// TIA Portal V17 export
// export: Created 2022-07-28T18:03:18.4124527Z, ExportSetting None, DisplayName Totally Integrated Automation Portal, DisplayVersion V17, DisplayName TIA Portal Openness, DisplayVersion V17, DisplayName TIA Portal Teamcenter Gateway, DisplayVersion V17, DisplayName TIA Portal Version Control Interface, DisplayVersion V17, DisplayName TIA Portal Test Suite Advanced, DisplayVersion V17, DisplayName SINAMICS Startdrive Advanced, DisplayVersion V17, DisplayName SINAMICS DCC, DisplayVersion V17, DisplayName SINAMICS Startdrive G130, G150, S120, S150, SINAMICS MV, S210, DisplayVersion V17, DisplayName SINAMICS Startdrive G110M, G120, G120C, G120D, G120P, G115D, DisplayVersion V17, DisplayName STEP 7 Professional, DisplayVersion V17, DisplayName SIMATIC Energy Suite, DisplayVersion V17, DisplayName STEP 7 CFC, DisplayVersion V17, DisplayName STEP 7 Safety, DisplayVersion V17, DisplayName WinCC Advanced / Unified PC, DisplayVersion V17, DisplayName SIMATIC Visualization Architect, DisplayVersion V17
TYPE "_ASensor_AlarmBits"
   STRUCT
      ErrorHH { ExternalAccessible := 'False'; ExternalVisible := 'False'; ExternalWritable := 'False'} : Bool;   // x0 - HH fault is active
      ErrorH { ExternalAccessible := 'False'; ExternalVisible := 'False'; ExternalWritable := 'False'} : Bool;   // x1 - H fault is active
      ErrorL { ExternalAccessible := 'False'; ExternalVisible := 'False'; ExternalWritable := 'False'} : Bool;   // x2 - L fault is active
      ErrorLL { ExternalAccessible := 'False'; ExternalVisible := 'False'; ExternalWritable := 'False'} : Bool;   // x3 - LL fault is active
      ErrorOvershoot { ExternalAccessible := 'False'; ExternalVisible := 'False'; ExternalWritable := 'False'} : Bool;   // x4 - Overshoot is active (act val > Maxlim)
      ErrorHiLimit { ExternalAccessible := 'False'; ExternalVisible := 'False'; ExternalWritable := 'False'} : Bool;   // x5 - Exceeding the maximum
      ErrorLoLimit { ExternalAccessible := 'False'; ExternalVisible := 'False'; ExternalWritable := 'False'} : Bool;   // x6 - Exceeding the minimum
      SimMode { ExternalAccessible := 'False'; ExternalVisible := 'False'; ExternalWritable := 'False'} : Bool;   // x7 - Sim mode is active
      NotSimMode { ExternalAccessible := 'False'; ExternalVisible := 'False'; ExternalWritable := 'False'} : Bool := true;   // x8 - Sim mode disabled
      SupplyErr { ExternalAccessible := 'False'; ExternalVisible := 'False'; ExternalWritable := 'False'} : Bool;   // x9 - Error of supply
      AW1_bit10 { ExternalAccessible := 'False'; ExternalVisible := 'False'; ExternalWritable := 'False'} : Bool;   // x10 -
      AW1_bit11 { ExternalAccessible := 'False'; ExternalVisible := 'False'; ExternalWritable := 'False'} : Bool;   // x11 -
      AW1_bit12 { ExternalAccessible := 'False'; ExternalVisible := 'False'; ExternalWritable := 'False'} : Bool;   // x12 -
      AW1_bit13 { ExternalAccessible := 'False'; ExternalVisible := 'False'; ExternalWritable := 'False'} : Bool;   // x13 -
      AW1_bit14 { ExternalAccessible := 'False'; ExternalVisible := 'False'; ExternalWritable := 'False'} : Bool;   // x14 -
      AW1_bit15 { ExternalAccessible := 'False'; ExternalVisible := 'False'; ExternalWritable := 'False'} : Bool;   // x15 - Not used
      DisableHH { ExternalAccessible := 'False'; ExternalVisible := 'False'; ExternalWritable := 'False'} : Bool;   // x0 - Disable HH fault detection
      DisableH { ExternalAccessible := 'False'; ExternalVisible := 'False'; ExternalWritable := 'False'} : Bool;   // x1 - Disable H fault detection
      DisableL { ExternalAccessible := 'False'; ExternalVisible := 'False'; ExternalWritable := 'False'} : Bool;   // x2 - Disable L fault detection
      DisableLL { ExternalAccessible := 'False'; ExternalVisible := 'False'; ExternalWritable := 'False'} : Bool;   // x3 - Disable LL fault detection
      SuppressedHH { ExternalAccessible := 'False'; ExternalVisible := 'False'; ExternalWritable := 'False'} : Bool;   // x4 - Suppress faults. HH
      SuppressedH { ExternalAccessible := 'False'; ExternalVisible := 'False'; ExternalWritable := 'False'} : Bool;   // x5 - Suppress faults. H
      SuppressedL { ExternalAccessible := 'False'; ExternalVisible := 'False'; ExternalWritable := 'False'} : Bool;   // x6 - Suppress faults. L
      SuppressedLL { ExternalAccessible := 'False'; ExternalVisible := 'False'; ExternalWritable := 'False'} : Bool;   // x7 - Suppress faults. LL
      DispWholeRange { ExternalAccessible := 'False'; ExternalVisible := 'False'; ExternalWritable := 'False'} : Bool;   // x8 - Display whole range
      DispWholPerc { ExternalAccessible := 'False'; ExternalVisible := 'False'; ExternalWritable := 'False'} : Bool;   // x9 - Display whole range (percents)
      DispPartRange { ExternalAccessible := 'False'; ExternalVisible := 'False'; ExternalWritable := 'False'} : Bool;   // x10 - Display a part of range
      DispPartPerc { ExternalAccessible := 'False'; ExternalVisible := 'False'; ExternalWritable := 'False'} : Bool;   // x11 - Display a part of range (percents)
      AW2_bit12 { ExternalAccessible := 'False'; ExternalVisible := 'False'; ExternalWritable := 'False'} : Bool;   // x12 -
      AW2_bit13 { ExternalAccessible := 'False'; ExternalVisible := 'False'; ExternalWritable := 'False'} : Bool;   // x13 -
      AW2_bit14 { ExternalAccessible := 'False'; ExternalVisible := 'False'; ExternalWritable := 'False'} : Bool;   // x14 -
      AW2_bit15 { ExternalAccessible := 'False'; ExternalVisible := 'False'; ExternalWritable := 'False'} : Bool;   // x15 - Not used
      EnableHH { ExternalAccessible := 'False'; ExternalVisible := 'False'; ExternalWritable := 'False'} : Bool;   // x0 - Enable/disable faults detection. HH
      EnableH { ExternalAccessible := 'False'; ExternalVisible := 'False'; ExternalWritable := 'False'} : Bool;   // x1 - Enable/disable faults detection. H
      EnableL { ExternalAccessible := 'False'; ExternalVisible := 'False'; ExternalWritable := 'False'} : Bool;   // x2 - Enable/disable faults detection. L
      EnableLL { ExternalAccessible := 'False'; ExternalVisible := 'False'; ExternalWritable := 'False'} : Bool;   // x3 - Enable/disable faults detection. LL
      ConsiderHH { ExternalAccessible := 'False'; ExternalVisible := 'False'; ExternalWritable := 'False'} : Bool;   // x4 - Consider HH fault
      ConsiderH { ExternalAccessible := 'False'; ExternalVisible := 'False'; ExternalWritable := 'False'} : Bool;   // x5 - Consider H fault
      ConsiderL { ExternalAccessible := 'False'; ExternalVisible := 'False'; ExternalWritable := 'False'} : Bool;   // x6 - Consider L fault
      ConsiderLL { ExternalAccessible := 'False'; ExternalVisible := 'False'; ExternalWritable := 'False'} : Bool;   // x7 - Consider LL fault
      AW3_bit8 { ExternalAccessible := 'False'; ExternalVisible := 'False'; ExternalWritable := 'False'} : Bool;   // x8 -
      AW3_bit9 { ExternalAccessible := 'False'; ExternalVisible := 'False'; ExternalWritable := 'False'} : Bool;   // x9 -
      AW3_bit10 { ExternalAccessible := 'False'; ExternalVisible := 'False'; ExternalWritable := 'False'} : Bool;   // x10 -
      AW3_bit11 { ExternalAccessible := 'False'; ExternalVisible := 'False'; ExternalWritable := 'False'} : Bool;   // x11 -
      AW3_bit12 { ExternalAccessible := 'False'; ExternalVisible := 'False'; ExternalWritable := 'False'} : Bool;   // x12 -
      AW3_bit13 { ExternalAccessible := 'False'; ExternalVisible := 'False'; ExternalWritable := 'False'} : Bool;   // x13 -
      AW3_bit14 { ExternalAccessible := 'False'; ExternalVisible := 'False'; ExternalWritable := 'False'} : Bool;   // x14 -
      AW3_bit15 { ExternalAccessible := 'False'; ExternalVisible := 'False'; ExternalWritable := 'False'} : Bool;   // x15 -
   END_STRUCT;
END_TYPE
